  60277 = '60277'
  60278 = '60278'
  60279 = '60279'
  60280 = '60280'
  60281 = '60281'
  60282 = '60282'
  60283 = '60283'
  60284 = '60284'
  60285 = '60285'
  60286 = '60286'
  60287 = '60287'
  60288 = '60288'
  60289 = '60289'
  60290 = '60290'
  60291 = '60291'
  60292 = '60292'
  60293 = '60293'
  60294 = '60294'
  60295 = '60295'
  60296 = '60296'
  60297 = '60297'
  60298 = '60298'
  60299 = '60299'
  60300 = '60300'
  60301 = '60301'
  60302 = '60302'
  60303 = '60303'
  60304 = '60304'
  60305 = '60305'
  60306 = '60306'
  60307 = '60307'
  60308 = '60308'
  60309 = '60309'
  60310 = '60310'
  60311 = '60311'
  60312 = '60312'
  60313 = '60313'
  60314 = '60314'
  60315 = '60315'
  60316 = '60316'
  60317 = '60317'
  60318 = '60318'
  60319 = '60319'
  60320 = '60320'
  60321 = '60321'
  60322 = '60322'
  60323 = '60323'
  60324 = '60324'
  60325 = '60325'
  60326 = '60326'
  60327 = '60327'
  60328 = '60328'
  60329 = '60329'
  60330 = '60330'
  60331 = '60331'
  60332 = '60332'
  60333 = '60333'
  60334 = '60334'
  60335 = '60335'
  60336 = '60336'
  60337 = '60337'
  60338 = '60338'
  60339 = '60339'
  60340 = '60340'
  60341 = '60341'
  60342 = '60342'
  60343 = '60343'
  60344 = '60344'
  60345 = '60345'
  60346 = '60346'
  60347 = '60347'
  60348 = '60348'
  60349 = '60349'
  60350 = '60350'
  60351 = '60351'
  60352 = '60352'
  60353 = '60353'
  60354 = '60354'
  60355 = '60355'
  60356 = '60356'
  60357 = '60357'
  60358 = '60358'
  60359 = '60359'
  60360 = '60360'
  60361 = '60361'
  60362 = '60362'
  60363 = '60363'
  60364 = '60364'
  60365 = '60365'
  60366 = '60366'
  60367 = '60367'
  60368 = '60368'
  60369 = '60369'
  60370 = '60370'
  60371 = '60371'
  60372 = '60372'
  60373 = '60373'
  60374 = '60374'
  60375 = '60375'
  60376 = '60376'
  60377 = '60377'
  60378 = '60378'
  60379 = '60379'
  60380 = '60380'
  60381 = '60381'
  60382 = '60382'
  60383 = '60383'
  60384 = '60384'
  60385 = '60385'
  60386 = '60386'
  60387 = '60387'
  60388 = '60388'
  60389 = '60389'
  60390 = '60390'
  60391 = '60391'
  60392 = '60392'
  60393 = '60393'
  60394 = '60394'
  60395 = '60395'
  60396 = '60396'
  60397 = '60397'
  60398 = '60398'
  60399 = '60399'
  60400 = '60400'
  60401 = '60401'
  60402 = '60402'
  60403 = '60403'
  60404 = '60404'
  60405 = '60405'
  60406 = '60406'
  60407 = '60407'
  60408 = '60408'
  60409 = '60409'
  60410 = '60410'
  60411 = '60411'
  60412 = '60412'
  60413 = '60413'
  60414 = '60414'
  60415 = '60415'
  60416 = '60416'
  60417 = '60417'
  60418 = '60418'
  60419 = '60419'
  60420 = '60420'
  60421 = '60421'
  60422 = '60422'
  60423 = '60423'
  60424 = '60424'
  60425 = '60425'
  60426 = '60426'
  60427 = '60427'
  60428 = '60428'
  60429 = '60429'
  60430 = '60430'
  60431 = '60431'
  60432 = '60432'
  60433 = '60433'
  60434 = '60434'
  60435 = '60435'
  60436 = '60436'
  60437 = '60437'
  60438 = '60438'
  60439 = '60439'
  60440 = '60440'
  60441 = '60441'
  60442 = '60442'
  60443 = '60443'
  60444 = '60444'
  60445 = '60445'
  60446 = '60446'
  60447 = '60447'
  60448 = '60448'
  60449 = '60449'
  60450 = '60450'
  60451 = '60451'
  60452 = '60452'
  60453 = '60453'
  60454 = '60454'
  60455 = '60455'
  60456 = '60456'
  60457 = '60457'
  60458 = '60458'
  60459 = '60459'
  60460 = '60460'
  60461 = '60461'
  60462 = '60462'
  60463 = '60463'
  60464 = '60464'
  60465 = '60465'
  60466 = '60466'
  60467 = '60467'
  60468 = '60468'
  60469 = '60469'
  60470 = '60470'
  60471 = '60471'
  60472 = '60472'
  60473 = '60473'
  60474 = '60474'
  60475 = '60475'
  60476 = '60476'
  60477 = '60477'
  60478 = '60478'
  60479 = '60479'
  60480 = '60480'
  60481 = '60481'
  60482 = '60482'
  60483 = '60483'
  60484 = '60484'
  60485 = '60485'
  60486 = '60486'
  60487 = '60487'
  60488 = '60488'
  60489 = '60489'
  60490 = '60490'
  60491 = '60491'
  60492 = '60492'
  60493 = '60493'
  60494 = '60494'
  60495 = '60495'
  60496 = '60496'
  60497 = '60497'
  60498 = '60498'
  60499 = '60499'
  60500 = '60500'
  60501 = '60501'
  60502 = '60502'
  60503 = '60503'
  60504 = '60504'
  60505 = '60505'
  60506 = '60506'
  60507 = '60507'
  60508 = '60508'
  60509 = '60509'
  60510 = '60510'
  60511 = '60511'
  60512 = '60512'
  60513 = '60513'
  60514 = '60514'
  60515 = '60515'
  60516 = '60516'
  60517 = '60517'
  60518 = '60518'
  60519 = '60519'
  60520 = '60520'
  60521 = '60521'
  60522 = '60522'
  60523 = '60523'
  60524 = '60524'
  60525 = '60525'
  60526 = '60526'
  60527 = '60527'
  60528 = '60528'
  60529 = '60529'
  60530 = '60530'
  60531 = '60531'
  60532 = '60532'
  60533 = '60533'
  60534 = '60534'
  60535 = '60535'
  60536 = '60536'
  60537 = '60537'
  60538 = '60538'
  60539 = '60539'
  60540 = '60540'
  60541 = '60541'
  60542 = '60542'
  60543 = '60543'
  60544 = '60544'
  60545 = '60545'
  60546 = '60546'
  60547 = '60547'
  60548 = '60548'
  60549 = '60549'
  60550 = '60550'
  60551 = '60551'
  60552 = '60552'
  60553 = '60553'
  60554 = '60554'
  60555 = '60555'
  60556 = '60556'
  60557 = '60557'
  60558 = '60558'
  60559 = '60559'
  60560 = '60560'
  60561 = '60561'
  60562 = '60562'
  60563 = '60563'
  60564 = '60564'
  60565 = '60565'
  60566 = '60566'
  60567 = '60567'
  60568 = '60568'
  60569 = '60569'
  60570 = '60570'
  60571 = '60571'
  60572 = '60572'
  60573 = '60573'
  60574 = '60574'
  60575 = '60575'
  60576 = '60576'
  60577 = '60577'
  60578 = '60578'
  60579 = '60579'
  60580 = '60580'
  60581 = '60581'
  60582 = '60582'
  60583 = '60583'
  60584 = '60584'
  60585 = '60585'
  60586 = '60586'
  60587 = '60587'
  60588 = '60588'
  60589 = '60589'
  60590 = '60590'
  60591 = '60591'
  60592 = '60592'
  60593 = '60593'
  60594 = '60594'
  60595 = '60595'
  60596 = '60596'
  60597 = '60597'
  60598 = '60598'
  60599 = '60599'
  60600 = '60600'
  60601 = '60601'
  60602 = '60602'
  60603 = '60603'
  60604 = '60604'
  60605 = '60605'
  60606 = '60606'
  60607 = '60607'
  60608 = '60608'
  60609 = '60609'
  60610 = '60610'
  60611 = '60611'
  60612 = '60612'
  60613 = '60613'
  60614 = '60614'
  60615 = '60615'
  60616 = '60616'
  60617 = '60617'
  60618 = '60618'
  60619 = '60619'
  60620 = '60620'
  60621 = '60621'
  60622 = '60622'
  60623 = '60623'
  60624 = '60624'
  60625 = '60625'
  60626 = '60626'
  60627 = '60627'
  60628 = '60628'
  60629 = '60629'
  60630 = '60630'
  60631 = '60631'
  60632 = '60632'
  60633 = '60633'
  60634 = '60634'
  60635 = '60635'
  60636 = '60636'
  60637 = '60637'
  60638 = '60638'
  60639 = '60639'
  60640 = '60640'
  60641 = '60641'
  60642 = '60642'
  60643 = '60643'
  60644 = '60644'
  60645 = '60645'
  60646 = '60646'
  60647 = '60647'
  60648 = '60648'
  60649 = '60649'
  60650 = '60650'
  60651 = '60651'
  60652 = '60652'
  60653 = '60653'
  60654 = '60654'
  60655 = '60655'
  60656 = '60656'
  60657 = '60657'
  60658 = '60658'
  60659 = '60659'
  60660 = '60660'
  60661 = '60661'
  60662 = '60662'
  60663 = '60663'
  60664 = '60664'
  60665 = '60665'
  60666 = '60666'
  60667 = '60667'
  60668 = '60668'
  60669 = '60669'
  60670 = '60670'
  60671 = '60671'
  60672 = '60672'
  60673 = '60673'
  60674 = '60674'
  60675 = '60675'
  60676 = '60676'
  60677 = '60677'
  60678 = '60678'
  60679 = '60679'
  60680 = '60680'
  60681 = '60681'
  60682 = '60682'
  60683 = '60683'
  60684 = '60684'
  60685 = '60685'
  60686 = '60686'
  60687 = '60687'
  60688 = '60688'
  60689 = '60689'
  60690 = '60690'
  60691 = '60691'
  60692 = '60692'
  60693 = '60693'
  60694 = '60694'
  60695 = '60695'
  60696 = '60696'
  60697 = '60697'
  60698 = '60698'
  60699 = '60699'
  60700 = '60700'
  60701 = '60701'
  60702 = '60702'
  60703 = '60703'
  60704 = '60704'
  60705 = '60705'
  60706 = '60706'
  60707 = '60707'
  60708 = '60708'
  60709 = '60709'
  60710 = '60710'
  60711 = '60711'
  60712 = '60712'
  60713 = '60713'
  60714 = '60714'
  60715 = '60715'
  60716 = '60716'
  60717 = '60717'
  60718 = '60718'
  60719 = '60719'
  60720 = '60720'
  60721 = '60721'
  60722 = '60722'
  60723 = '60723'
  60724 = '60724'
  60725 = '60725'
  60726 = '60726'
  60727 = '60727'
  60728 = '60728'
  60729 = '60729'
  60730 = '60730'
  60731 = '60731'
  60732 = '60732'
  60733 = '60733'
  60734 = '60734'
  60735 = '60735'
  60736 = '60736'
  60737 = '60737'
  60738 = '60738'
  60739 = '60739'
  60740 = '60740'
  60741 = '60741'
  60742 = '60742'
  60743 = '60743'
  60744 = '60744'
  60745 = '60745'
  60746 = '60746'
  60747 = '60747'
  60748 = '60748'
  60749 = '60749'
  60750 = '60750'
  60751 = '60751'
  60752 = '60752'
  60753 = '60753'
  60754 = '60754'
  60755 = '60755'
  60756 = '60756'
  60757 = '60757'
  60758 = '60758'
  60759 = '60759'
  60760 = '60760'
  60761 = '60761'
  60762 = '60762'
  60763 = '60763'
  60764 = '60764'
  60765 = '60765'
  60766 = '60766'
  60767 = '60767'
  60768 = '60768'
  60769 = '60769'
  60770 = '60770'
  60771 = '60771'
  60772 = '60772'
  60773 = '60773'
  60774 = '60774'
  60775 = '60775'
  60776 = '60776'
  60777 = '60777'
  60778 = '60778'
  60779 = '60779'
  60780 = '60780'
  60781 = '60781'
  60782 = '60782'
  60783 = '60783'
  60784 = '60784'
  60785 = '60785'
  60786 = '60786'
  60787 = '60787'
  60788 = '60788'
  60789 = '60789'
  60790 = '60790'
  60791 = '60791'
  60792 = '60792'
  60793 = '60793'
  60794 = '60794'
  60795 = '60795'
  60796 = '60796'
  60797 = '60797'
  60798 = '60798'
  60799 = '60799'
  60800 = '60800'
  60801 = '60801'
  60802 = '60802'
  60803 = '60803'
  60804 = '60804'
  60805 = '60805'
  60806 = '60806'
  60807 = '60807'
  60808 = '60808'
  60809 = '60809'
  60810 = '60810'
  60811 = '60811'
  60812 = '60812'
  60813 = '60813'
  60814 = '60814'
  60815 = '60815'
  60816 = '60816'
  60817 = '60817'
  60818 = '60818'
  60819 = '60819'
  60820 = '60820'
  60821 = '60821'
  60822 = '60822'
  60823 = '60823'
  60824 = '60824'
  60825 = '60825'
  60826 = '60826'
  60827 = '60827'
  60828 = '60828'
  60829 = '60829'
  60830 = '60830'
  60831 = '60831'
  60832 = '60832'
  60833 = '60833'
  60834 = '60834'
  60835 = '60835'
  60836 = '60836'
  60837 = '60837'
  60838 = '60838'
  60839 = '60839'
  60840 = '60840'
  60841 = '60841'
  60842 = '60842'
  60843 = '60843'
  60844 = '60844'
  60845 = '60845'
  60846 = '60846'
  60847 = '60847'
  60848 = '60848'
  60849 = '60849'
  60850 = '60850'
  60851 = '60851'
  60852 = '60852'
  60853 = '60853'
  60854 = '60854'
  60855 = '60855'
  60856 = '60856'
  60857 = '60857'
  60858 = '60858'
  60859 = '60859'
  60860 = '60860'
  60861 = '60861'
  60862 = '60862'
  60863 = '60863'
  60864 = '60864'
  60865 = '60865'
  60866 = '60866'
  60867 = '60867'
  60868 = '60868'
  60869 = '60869'
  60870 = '60870'
  60871 = '60871'
  60872 = '60872'
  60873 = '60873'
  60874 = '60874'
  60875 = '60875'
  60876 = '60876'
  60877 = '60877'
  60878 = '60878'
  60879 = '60879'
  60880 = '60880'
  60881 = '60881'
  60882 = '60882'
  60883 = '60883'
  60884 = '60884'
  60885 = '60885'
  60886 = '60886'
  60887 = '60887'
  60888 = '60888'
  60889 = '60889'
  60890 = '60890'
  60891 = '60891'
  60892 = '60892'
  60893 = '60893'
  60894 = '60894'
  60895 = '60895'
  60896 = '60896'
  60897 = '60897'
  60898 = '60898'
  60899 = '60899'
  60900 = '60900'
  60901 = '60901'
  60902 = '60902'
  60903 = '60903'
  60904 = '60904'
  60905 = '60905'
  60906 = '60906'
  60907 = '60907'
  60908 = '60908'
  60909 = '60909'
  60910 = '60910'
  60911 = '60911'
  60912 = '60912'
  60913 = '60913'
  60914 = '60914'
  60915 = '60915'
  60916 = '60916'
  60917 = '60917'
  60918 = '60918'
  60919 = '60919'
  60920 = '60920'
  60921 = '60921'
  60922 = '60922'
  60923 = '60923'
  60924 = '60924'
  60925 = '60925'
  60926 = '60926'
  60927 = '60927'
  60928 = '60928'
  60929 = '60929'
  60930 = '60930'
  60931 = '60931'
  60932 = '60932'
  60933 = '60933'
  60934 = '60934'
  60935 = '60935'
  60936 = '60936'
  60937 = '60937'
  60938 = '60938'
  60939 = '60939'
  60940 = '60940'
  60941 = '60941'
  60942 = '60942'
  60943 = '60943'
  60944 = '60944'
  60945 = '60945'
  60946 = '60946'
  60947 = '60947'
  60948 = '60948'
  60949 = '60949'
  60950 = '60950'
  60951 = '60951'
  60952 = '60952'
  60953 = '60953'
  60954 = '60954'
  60955 = '60955'
  60956 = '60956'
  60957 = '60957'
  60958 = '60958'
  60959 = '60959'
  60960 = '60960'
  60961 = '60961'
  60962 = '60962'
  60963 = '60963'
  60964 = '60964'
  60965 = '60965'
  60966 = '60966'
  60967 = '60967'
  60968 = '60968'
  60969 = '60969'
  60970 = '60970'
  60971 = '60971'
  60972 = '60972'
  60973 = '60973'
  60974 = '60974'
  60975 = '60975'
  60976 = '60976'
  60977 = '60977'
  60978 = '60978'
  60979 = '60979'
  60980 = '60980'
  60981 = '60981'
  60982 = '60982'
  60983 = '60983'
  60984 = '60984'
  60985 = '60985'
  60986 = '60986'
  60987 = '60987'
  60988 = '60988'
  60989 = '60989'
  60990 = '60990'
  60991 = '60991'
  60992 = '60992'
  60993 = '60993'
  60994 = '60994'
  60995 = '60995'
  60996 = '60996'
  60997 = '60997'
  60998 = '60998'
  60999 = '60999'
  61000 = '61000'
  61001 = '61001'
  61002 = '61002'
  61003 = '61003'
  61004 = '61004'
  61005 = '61005'
  61006 = '61006'
  61007 = '61007'
  61008 = '61008'
  61009 = '61009'
  61010 = '61010'
  61011 = '61011'
  61012 = '61012'
  61013 = '61013'
  61014 = '61014'
  61015 = '61015'
  61016 = '61016'
  61017 = '61017'
  61018 = '61018'
  61019 = '61019'
  61020 = '61020'
  61021 = '61021'
  61022 = '61022'
  61023 = '61023'
  61024 = '61024'
  61025 = '61025'
  61026 = '61026'
  61027 = '61027'
  61028 = '61028'
  61029 = '61029'
  61030 = '61030'
  61031 = '61031'
  61032 = '61032'
  61033 = '61033'
  61034 = '61034'
  61035 = '61035'
  61036 = '61036'
  61037 = '61037'
  61038 = '61038'
  61039 = '61039'
  61040 = '61040'
  61041 = '61041'
  61042 = '61042'
  61043 = '61043'
  61044 = '61044'
  61045 = '61045'
  61046 = '61046'
  61047 = '61047'
  61048 = '61048'
  61049 = '61049'
  61050 = '61050'
  61051 = '61051'
  61052 = '61052'
  61053 = '61053'
  61054 = '61054'
  61055 = '61055'
  61056 = '61056'
  61057 = '61057'
  61058 = '61058'
  61059 = '61059'
  61060 = '61060'
  61061 = '61061'
  61062 = '61062'
  61063 = '61063'
  61064 = '61064'
  61065 = '61065'
  61066 = '61066'
  61067 = '61067'
  61068 = '61068'
  61069 = '61069'
  61070 = '61070'
  61071 = '61071'
  61072 = '61072'
  61073 = '61073'
  61074 = '61074'
  61075 = '61075'
  61076 = '61076'
  61077 = '61077'
  61078 = '61078'
  61079 = '61079'
  61080 = '61080'
  61081 = '61081'
  61082 = '61082'
  61083 = '61083'
  61084 = '61084'
  61085 = '61085'
  61086 = '61086'
  61087 = '61087'
  61088 = '61088'
  61089 = '61089'
  61090 = '61090'
  61091 = '61091'
  61092 = '61092'
  61093 = '61093'
  61094 = '61094'
  61095 = '61095'
  61096 = '61096'
  61097 = '61097'
  61098 = '61098'
  61099 = '61099'
  61100 = '61100'
  61101 = '61101'
  61102 = '61102'
  61103 = '61103'
  61104 = '61104'
  61105 = '61105'
  61106 = '61106'
  61107 = '61107'
  61108 = '61108'
  61109 = '61109'
  61110 = '61110'
  61111 = '61111'
  61112 = '61112'
  61113 = '61113'
  61114 = '61114'
  61115 = '61115'
  61116 = '61116'
  61117 = '61117'
  61118 = '61118'
  61119 = '61119'
  61120 = '61120'
  61121 = '61121'
  61122 = '61122'
  61123 = '61123'
  61124 = '61124'
  61125 = '61125'
  61126 = '61126'
  61127 = '61127'
  61128 = '61128'
  61129 = '61129'
  61130 = '61130'
  61131 = '61131'
  61132 = '61132'
  61133 = '61133'
  61134 = '61134'
  61135 = '61135'
  61136 = '61136'
  61137 = '61137'
  61138 = '61138'
  61139 = '61139'
  61140 = '61140'
  61141 = '61141'
  61142 = '61142'
  61143 = '61143'
  61144 = '61144'
  61145 = '61145'
  61146 = '61146'
  61147 = '61147'
  61148 = '61148'
  61149 = '61149'
  61150 = '61150'
  61151 = '61151'
  61152 = '61152'
  61153 = '61153'
  61154 = '61154'
  61155 = '61155'
  61156 = '61156'
  61157 = '61157'
  61158 = '61158'
  61159 = '61159'
  61160 = '61160'
  61161 = '61161'
  61162 = '61162'
  61163 = '61163'
  61164 = '61164'
  61165 = '61165'
  61166 = '61166'
  61167 = '61167'
  61168 = '61168'
  61169 = '61169'
  61170 = '61170'
  61171 = '61171'
  61172 = '61172'
  61173 = '61173'
  61174 = '61174'
  61175 = '61175'
  61176 = '61176'
  61177 = '61177'
  61178 = '61178'
  61179 = '61179'
  61180 = '61180'
  61181 = '61181'
  61182 = '61182'
  61183 = '61183'
  61184 = '61184'
  61185 = '61185'
  61186 = '61186'
  61187 = '61187'
  61188 = '61188'
  61189 = '61189'
  61190 = '61190'
  61191 = '61191'
  61192 = '61192'
  61193 = '61193'
  61194 = '61194'
  61195 = '61195'
  61196 = '61196'
  61197 = '61197'
  61198 = '61198'
  61199 = '61199'
  61200 = '61200'
  61201 = '61201'
  61202 = '61202'
  61203 = '61203'
  61204 = '61204'
  61205 = '61205'
  61206 = '61206'
  61207 = '61207'
  61208 = '61208'
  61209 = '61209'
  61210 = '61210'
  61211 = '61211'
  61212 = '61212'
  61213 = '61213'
  61214 = '61214'
  61215 = '61215'
  61216 = '61216'
  61217 = '61217'
  61218 = '61218'
  61219 = '61219'
  61220 = '61220'
  61221 = '61221'
  61222 = '61222'
  61223 = '61223'
  61224 = '61224'
  61225 = '61225'
  61226 = '61226'
  61227 = '61227'
  61228 = '61228'
  61229 = '61229'
  61230 = '61230'
  61231 = '61231'
  61232 = '61232'
  61233 = '61233'
  61234 = '61234'
  61235 = '61235'
  61236 = '61236'
  61237 = '61237'
  61238 = '61238'
  61239 = '61239'
  61240 = '61240'
  61241 = '61241'
  61242 = '61242'
  61243 = '61243'
  61244 = '61244'
  61245 = '61245'
  61246 = '61246'
  61247 = '61247'
  61248 = '61248'
  61249 = '61249'
  61250 = '61250'
  61251 = '61251'
  61252 = '61252'
  61253 = '61253'
  61254 = '61254'
  61255 = '61255'
  61256 = '61256'
  61257 = '61257'
  61258 = '61258'
  61259 = '61259'
  61260 = '61260'
  61261 = '61261'
  61262 = '61262'
  61263 = '61263'
  61264 = '61264'
  61265 = '61265'
  61266 = '61266'
  61267 = '61267'
  61268 = '61268'
  61269 = '61269'
  61270 = '61270'
  61271 = '61271'
  61272 = '61272'
  61273 = '61273'
  61274 = '61274'
  61275 = '61275'
  61276 = '61276'
  61277 = '61277'
  61278 = '61278'
  61279 = '61279'
  61280 = '61280'
  61281 = '61281'
  61282 = '61282'
  61283 = '61283'
  61284 = '61284'
  61285 = '61285'
  61286 = '61286'
  61287 = '61287'
  61288 = '61288'
  61289 = '61289'
  61290 = '61290'
  61291 = '61291'
  61292 = '61292'
  61293 = '61293'
  61294 = '61294'
  61295 = '61295'
  61296 = '61296'
  61297 = '61297'
  61298 = '61298'
  61299 = '61299'
  61300 = '61300'
  61301 = '61301'
  61302 = '61302'
  61303 = '61303'
  61304 = '61304'
  61305 = '61305'
  61306 = '61306'
  61307 = '61307'
  61308 = '61308'
  61309 = '61309'
  61310 = '61310'
  61311 = '61311'
  61312 = '61312'
  61313 = '61313'
  61314 = '61314'
  61315 = '61315'
  61316 = '61316'
  61317 = '61317'
  61318 = '61318'
  61319 = '61319'
  61320 = '61320'
  61321 = '61321'
  61322 = '61322'
  61323 = '61323'
  61324 = '61324'
  61325 = '61325'
  61326 = '61326'
  61327 = '61327'
  61328 = '61328'
  61329 = '61329'
  61330 = '61330'
  61331 = '61331'
  61332 = '61332'
  61333 = '61333'
  61334 = '61334'
  61335 = '61335'
  61336 = '61336'
  61337 = '61337'
  61338 = '61338'
  61339 = '61339'
  61340 = '61340'
  61341 = '61341'
  61342 = '61342'
  61343 = '61343'
  61344 = '61344'
  61345 = '61345'
  61346 = '61346'
  61347 = '61347'
  61348 = '61348'
  61349 = '61349'
  61350 = '61350'
  61351 = '61351'
  61352 = '61352'
  61353 = '61353'
  61354 = '61354'
  61355 = '61355'
  61356 = '61356'
  61357 = '61357'
  61358 = '61358'
  61359 = '61359'
  61360 = '61360'
  61361 = '61361'
  61362 = '61362'
  61363 = '61363'
  61364 = '61364'
  61365 = '61365'
  61366 = '61366'
  61367 = '61367'
  61368 = '61368'
  61369 = '61369'
  61370 = '61370'
  61371 = '61371'
  61372 = '61372'
  61373 = '61373'
  61374 = '61374'
  61375 = '61375'
  61376 = '61376'
  61377 = '61377'
  61378 = '61378'
  61379 = '61379'
  61380 = '61380'
  61381 = '61381'
  61382 = '61382'
  61383 = '61383'
  61384 = '61384'
  61385 = '61385'
  61386 = '61386'
  61387 = '61387'
  61388 = '61388'
  61389 = '61389'
  61390 = '61390'
  61391 = '61391'
  61392 = '61392'
  61393 = '61393'
  61394 = '61394'
  61395 = '61395'
  61396 = '61396'
  61397 = '61397'
  61398 = '61398'
  61399 = '61399'
  61400 = '61400'
  61401 = '61401'
  61402 = '61402'
  61403 = '61403'
  61404 = '61404'
  61405 = '61405'
  61406 = '61406'
  61407 = '61407'
  61408 = '61408'
  61409 = '61409'
  61410 = '61410'
  61411 = '61411'
  61412 = '61412'
  61413 = '61413'
  61414 = '61414'
  61415 = '61415'
  61416 = '61416'
  61417 = '61417'
  61418 = '61418'
  61419 = '61419'
  61420 = '61420'
  61421 = '61421'
  61422 = '61422'
  61423 = '61423'
  61424 = '61424'
  61425 = '61425'
  61426 = '61426'
  61427 = '61427'
  61428 = '61428'
  61429 = '61429'
  61430 = '61430'
  61431 = '61431'
  61432 = '61432'
  61433 = '61433'
  61434 = '61434'
  61435 = '61435'
  61436 = '61436'
  61437 = '61437'
  61438 = '61438'
  61439 = '61439'
  61440 = '61440'
  61441 = '61441'
  61442 = '61442'
  61443 = '61443'
  61444 = '61444'
  61445 = '61445'
  61446 = '61446'
  61447 = '61447'
  61448 = '61448'
  61449 = '61449'
  61450 = '61450'
  61451 = '61451'
  61452 = '61452'
  61453 = '61453'
  61454 = '61454'
  61455 = '61455'
  61456 = '61456'
  61457 = '61457'
  61458 = '61458'
  61459 = '61459'
  61460 = '61460'
  61461 = '61461'
  61462 = '61462'
  61463 = '61463'
  61464 = '61464'
  61465 = '61465'
  61466 = '61466'
  61467 = '61467'
  61468 = '61468'
  61469 = '61469'
  61470 = '61470'
  61471 = '61471'
  61472 = '61472'
  61473 = '61473'
  61474 = '61474'
  61475 = '61475'
  61476 = '61476'
  61477 = '61477'
  61478 = '61478'
  61479 = '61479'
  61480 = '61480'
  61481 = '61481'
  61482 = '61482'
  61483 = '61483'
  61484 = '61484'
  61485 = '61485'
  61486 = '61486'
  61487 = '61487'
  61488 = '61488'
  61489 = '61489'
  61490 = '61490'
  61491 = '61491'
  61492 = '61492'
  61493 = '61493'
  61494 = '61494'
  61495 = '61495'
  61496 = '61496'
  61497 = '61497'
  61498 = '61498'
  61499 = '61499'
  61500 = '61500'
  61501 = '61501'
  61502 = '61502'
  61503 = '61503'
  61504 = '61504'
  61505 = '61505'
  61506 = '61506'
  61507 = '61507'
  61508 = '61508'
  61509 = '61509'
  61510 = '61510'
  61511 = '61511'
  61512 = '61512'
  61513 = '61513'
  61514 = '61514'
  61515 = '61515'
  61516 = '61516'
  61517 = '61517'
  61518 = '61518'
  61519 = '61519'
  61520 = '61520'
  61521 = '61521'
  61522 = '61522'
  61523 = '61523'
  61524 = '61524'
  61525 = '61525'
  61526 = '61526'
  61527 = '61527'
  61528 = '61528'
  61529 = '61529'
  61530 = '61530'
  61531 = '61531'
  61532 = '61532'
  61533 = '61533'
  61534 = '61534'
  61535 = '61535'
  61536 = '61536'
  61537 = '61537'
  61538 = '61538'
  61539 = '61539'
  61540 = '61540'
  61541 = '61541'
  61542 = '61542'
  61543 = '61543'
  61544 = '61544'
  61545 = '61545'
  61546 = '61546'
  61547 = '61547'
  61548 = '61548'
  61549 = '61549'
  61550 = '61550'
  61551 = '61551'
  61552 = '61552'
  61553 = '61553'
  61554 = '61554'
  61555 = '61555'
  61556 = '61556'
  61557 = '61557'
  61558 = '61558'
  61559 = '61559'
  61560 = '61560'
  61561 = '61561'
  61562 = '61562'
  61563 = '61563'
  61564 = '61564'
  61565 = '61565'
  61566 = '61566'
  61567 = '61567'
  61568 = '61568'
  61569 = '61569'
  61570 = '61570'
  61571 = '61571'
  61572 = '61572'
  61573 = '61573'
  61574 = '61574'
  61575 = '61575'
  61576 = '61576'
  61577 = '61577'
  61578 = '61578'
  61579 = '61579'
  61580 = '61580'
  61581 = '61581'
  61582 = '61582'
  61583 = '61583'
  61584 = '61584'
  61585 = '61585'
  61586 = '61586'
  61587 = '61587'
  61588 = '61588'
  61589 = '61589'
  61590 = '61590'
  61591 = '61591'
  61592 = '61592'
  61593 = '61593'
  61594 = '61594'
  61595 = '61595'
  61596 = '61596'
  61597 = '61597'
  61598 = '61598'
  61599 = '61599'
  61600 = '61600'
  61601 = '61601'
  61602 = '61602'
  61603 = '61603'
  61604 = '61604'
  61605 = '61605'
  61606 = '61606'
  61607 = '61607'
  61608 = '61608'
  61609 = '61609'
  61610 = '61610'
  61611 = '61611'
  61612 = '61612'
  61613 = '61613'
  61614 = '61614'
  61615 = '61615'
  61616 = '61616'
  61617 = '61617'
  61618 = '61618'
  61619 = '61619'
  61620 = '61620'
  61621 = '61621'
  61622 = '61622'
  61623 = '61623'
  61624 = '61624'
  61625 = '61625'
  61626 = '61626'
  61627 = '61627'
  61628 = '61628'
  61629 = '61629'
  61630 = '61630'
  61631 = '61631'
  61632 = '61632'
  61633 = '61633'
  61634 = '61634'
  61635 = '61635'
  61636 = '61636'
  61637 = '61637'
  61638 = '61638'
  61639 = '61639'
  61640 = '61640'
  61641 = '61641'
  61642 = '61642'
  61643 = '61643'
  61644 = '61644'
  61645 = '61645'
  61646 = '61646'
  61647 = '61647'
  61648 = '61648'
  61649 = '61649'
  61650 = '61650'
  61651 = '61651'
  61652 = '61652'
  61653 = '61653'
  61654 = '61654'
  61655 = '61655'
  61656 = '61656'
  61657 = '61657'
  61658 = '61658'
  61659 = '61659'
  61660 = '61660'
  61661 = '61661'
  61662 = '61662'
  61663 = '61663'
  61664 = '61664'
  61665 = '61665'
  61666 = '61666'
  61667 = '61667'
  61668 = '61668'
  61669 = '61669'
  61670 = '61670'
  61671 = '61671'
  61672 = '61672'
  61673 = '61673'
  61674 = '61674'
  61675 = '61675'
  61676 = '61676'
  61677 = '61677'
  61678 = '61678'
  61679 = '61679'
  61680 = '61680'
  61681 = '61681'
  61682 = '61682'
  61683 = '61683'
  61684 = '61684'
  61685 = '61685'
  61686 = '61686'
  61687 = '61687'
  61688 = '61688'
  61689 = '61689'
  61690 = '61690'
  61691 = '61691'
  61692 = '61692'
  61693 = '61693'
  61694 = '61694'
  61695 = '61695'
  61696 = '61696'
  61697 = '61697'
  61698 = '61698'
  61699 = '61699'
  61700 = '61700'
  61701 = '61701'
  61702 = '61702'
  61703 = '61703'
  61704 = '61704'
  61705 = '61705'
  61706 = '61706'
  61707 = '61707'
  61708 = '61708'
  61709 = '61709'
  61710 = '61710'
  61711 = '61711'
  61712 = '61712'
  61713 = '61713'
  61714 = '61714'
  61715 = '61715'
  61716 = '61716'
  61717 = '61717'
  61718 = '61718'
  61719 = '61719'
  61720 = '61720'
  61721 = '61721'
  61722 = '61722'
  61723 = '61723'
  61724 = '61724'
  61725 = '61725'
  61726 = '61726'
  61727 = '61727'
  61728 = '61728'
  61729 = '61729'
  61730 = '61730'
  61731 = '61731'
  61732 = '61732'
  61733 = '61733'
  61734 = '61734'
  61735 = '61735'
  61736 = '61736'
  61737 = '61737'
  61738 = '61738'
  61739 = '61739'
  61740 = '61740'
  61741 = '61741'
  61742 = '61742'
  61743 = '61743'
  61744 = '61744'
  61745 = '61745'
  61746 = '61746'
  61747 = '61747'
  61748 = '61748'
  61749 = '61749'
  61750 = '61750'
  61751 = '61751'
  61752 = '61752'
  61753 = '61753'
  61754 = '61754'
  61755 = '61755'
  61756 = '61756'
  61757 = '61757'
  61758 = '61758'
  61759 = '61759'
  61760 = '61760'
  61761 = '61761'
  61762 = '61762'
  61763 = '61763'
  61764 = '61764'
  61765 = '61765'
  61766 = '61766'
  61767 = '61767'
  61768 = '61768'
  61769 = '61769'
  61770 = '61770'
  61771 = '61771'
  61772 = '61772'
  61773 = '61773'
  61774 = '61774'
  61775 = '61775'
  61776 = '61776'
  61777 = '61777'
  61778 = '61778'
  61779 = '61779'
  61780 = '61780'
  61781 = '61781'
  61782 = '61782'
  61783 = '61783'
  61784 = '61784'
  61785 = '61785'
  61786 = '61786'
  61787 = '61787'
  61788 = '61788'
  61789 = '61789'
  61790 = '61790'
  61791 = '61791'
  61792 = '61792'
  61793 = '61793'
  61794 = '61794'
  61795 = '61795'
  61796 = '61796'
  61797 = '61797'
  61798 = '61798'
  61799 = '61799'
  61800 = '61800'
  61801 = '61801'
  61802 = '61802'
  61803 = '61803'
  61804 = '61804'
  61805 = '61805'
  61806 = '61806'
  61807 = '61807'
  61808 = '61808'
  61809 = '61809'
  61810 = '61810'
  61811 = '61811'
  61812 = '61812'
  61813 = '61813'
  61814 = '61814'
  61815 = '61815'
  61816 = '61816'
  61817 = '61817'
  61818 = '61818'
  61819 = '61819'
  61820 = '61820'
  61821 = '61821'
  61822 = '61822'
  61823 = '61823'
  61824 = '61824'
  61825 = '61825'
  61826 = '61826'
  61827 = '61827'
  61828 = '61828'
  61829 = '61829'
  61830 = '61830'
  61831 = '61831'
  61832 = '61832'
  61833 = '61833'
  61834 = '61834'
  61835 = '61835'
  61836 = '61836'
  61837 = '61837'
  61838 = '61838'
  61839 = '61839'
  61840 = '61840'
  61841 = '61841'
  61842 = '61842'
  61843 = '61843'
  61844 = '61844'
  61845 = '61845'
  61846 = '61846'
  61847 = '61847'
  61848 = '61848'
  61849 = '61849'
  61850 = '61850'
  61851 = '61851'
  61852 = '61852'
  61853 = '61853'
  61854 = '61854'
  61855 = '61855'
  61856 = '61856'
  61857 = '61857'
  61858 = '61858'
  61859 = '61859'
  61860 = '61860'
  61861 = '61861'
  61862 = '61862'
  61863 = '61863'
  61864 = '61864'
  61865 = '61865'
  61866 = '61866'
  61867 = '61867'
  61868 = '61868'
  61869 = '61869'
  61870 = '61870'
  61871 = '61871'
  61872 = '61872'
  61873 = '61873'
  61874 = '61874'
  61875 = '61875'
  61876 = '61876'
  61877 = '61877'
  61878 = '61878'
  61879 = '61879'
  61880 = '61880'
  61881 = '61881'
  61882 = '61882'
  61883 = '61883'
  61884 = '61884'
  61885 = '61885'
  61886 = '61886'
  61887 = '61887'
  61888 = '61888'
  61889 = '61889'
  61890 = '61890'
  61891 = '61891'
  61892 = '61892'
  61893 = '61893'
  61894 = '61894'
  61895 = '61895'
  61896 = '61896'
  61897 = '61897'
  61898 = '61898'
  61899 = '61899'
  61900 = '61900'
  61901 = '61901'
  61902 = '61902'
  61903 = '61903'
  61904 = '61904'
  61905 = '61905'
  61906 = '61906'
  61907 = '61907'
  61908 = '61908'
  61909 = '61909'
  61910 = '61910'
  61911 = '61911'
  61912 = '61912'
  61913 = '61913'
  61914 = '61914'
  61915 = '61915'
  61916 = '61916'
  61917 = '61917'
  61918 = '61918'
  61919 = '61919'
  61920 = '61920'
  61921 = '61921'
  61922 = '61922'
  61923 = '61923'
  61924 = '61924'
  61925 = '61925'
  61926 = '61926'
  61927 = '61927'
  61928 = '61928'
  61929 = '61929'
  61930 = '61930'
  61931 = '61931'
  61932 = '61932'
  61933 = '61933'
  61934 = '61934'
  61935 = '61935'
  61936 = '61936'
  61937 = '61937'
  61938 = '61938'
  61939 = '61939'
  61940 = '61940'
  61941 = '61941'
  61942 = '61942'
  61943 = '61943'
  61944 = '61944'
  61945 = '61945'
  61946 = '61946'
  61947 = '61947'
  61948 = '61948'
  61949 = '61949'
  61950 = '61950'
  61951 = '61951'
  61952 = '61952'
  61953 = '61953'
  61954 = '61954'
  61955 = '61955'
  61956 = '61956'
  61957 = '61957'
  61958 = '61958'
  61959 = '61959'
  61960 = '61960'
  61961 = '61961'
  61962 = '61962'
  61963 = '61963'
  61964 = '61964'
  61965 = '61965'
  61966 = '61966'
  61967 = '61967'
  61968 = '61968'
  61969 = '61969'
  61970 = '61970'
  61971 = '61971'
  61972 = '61972'
  61973 = '61973'
  61974 = '61974'
  61975 = '61975'
  61976 = '61976'
  61977 = '61977'
  61978 = '61978'
  61979 = '61979'
  61980 = '61980'
  61981 = '61981'
  61982 = '61982'
  61983 = '61983'
  61984 = '61984'
  61985 = '61985'
  61986 = '61986'
  61987 = '61987'
  61988 = '61988'
  61989 = '61989'
  61990 = '61990'
  61991 = '61991'
  61992 = '61992'
  61993 = '61993'
  61994 = '61994'
  61995 = '61995'
  61996 = '61996'
  61997 = '61997'
  61998 = '61998'
  61999 = '61999'
  62000 = '62000'
  62001 = '62001'
  62002 = '62002'
  62003 = '62003'
  62004 = '62004'
  62005 = '62005'
  62006 = '62006'
  62007 = '62007'
  62008 = '62008'
  62009 = '62009'
  62010 = '62010'
  62011 = '62011'
  62012 = '62012'
  62013 = '62013'
  62014 = '62014'
  62015 = '62015'
  62016 = '62016'
  62017 = '62017'
  62018 = '62018'
  62019 = '62019'
  62020 = '62020'
  62021 = '62021'
  62022 = '62022'
  62023 = '62023'
  62024 = '62024'
  62025 = '62025'
  62026 = '62026'
  62027 = '62027'
  62028 = '62028'
  62029 = '62029'
  62030 = '62030'
  62031 = '62031'
  62032 = '62032'
  62033 = '62033'
  62034 = '62034'
  62035 = '62035'
  62036 = '62036'
  62037 = '62037'
  62038 = '62038'
  62039 = '62039'
  62040 = '62040'
  62041 = '62041'
  62042 = '62042'
  62043 = '62043'
  62044 = '62044'
  62045 = '62045'
  62046 = '62046'
  62047 = '62047'
  62048 = '62048'
  62049 = '62049'
  62050 = '62050'
  62051 = '62051'
  62052 = '62052'
  62053 = '62053'
  62054 = '62054'
  62055 = '62055'
  62056 = '62056'
  62057 = '62057'
  62058 = '62058'
  62059 = '62059'
  62060 = '62060'
  62061 = '62061'
  62062 = '62062'
  62063 = '62063'
  62064 = '62064'
  62065 = '62065'
  62066 = '62066'
  62067 = '62067'
  62068 = '62068'
  62069 = '62069'
  62070 = '62070'
  62071 = '62071'
  62072 = '62072'
  62073 = '62073'
  62074 = '62074'
  62075 = '62075'
  62076 = '62076'
  62077 = '62077'
  62078 = '62078'
  62079 = '62079'
  62080 = '62080'
  62081 = '62081'
  62082 = '62082'
  62083 = '62083'
  62084 = '62084'
  62085 = '62085'
  62086 = '62086'
  62087 = '62087'
  62088 = '62088'
  62089 = '62089'
  62090 = '62090'
  62091 = '62091'
  62092 = '62092'
  62093 = '62093'
  62094 = '62094'
  62095 = '62095'
  62096 = '62096'
  62097 = '62097'
  62098 = '62098'
  62099 = '62099'
  62100 = '62100'
  62101 = '62101'
  62102 = '62102'
  62103 = '62103'
  62104 = '62104'
  62105 = '62105'
  62106 = '62106'
  62107 = '62107'
  62108 = '62108'
  62109 = '62109'
  62110 = '62110'
  62111 = '62111'
  62112 = '62112'
  62113 = '62113'
  62114 = '62114'
  62115 = '62115'
  62116 = '62116'
  62117 = '62117'
  62118 = '62118'
  62119 = '62119'
  62120 = '62120'
  62121 = '62121'
  62122 = '62122'
  62123 = '62123'
  62124 = '62124'
  62125 = '62125'
  62126 = '62126'
  62127 = '62127'
  62128 = '62128'
  62129 = '62129'
  62130 = '62130'
  62131 = '62131'
  62132 = '62132'
  62133 = '62133'
  62134 = '62134'
  62135 = '62135'
  62136 = '62136'
  62137 = '62137'
  62138 = '62138'
  62139 = '62139'
  62140 = '62140'
  62141 = '62141'
  62142 = '62142'
  62143 = '62143'
  62144 = '62144'
  62145 = '62145'
  62146 = '62146'
  62147 = '62147'
  62148 = '62148'
  62149 = '62149'
  62150 = '62150'
  62151 = '62151'
  62152 = '62152'
  62153 = '62153'
  62154 = '62154'
  62155 = '62155'
  62156 = '62156'
  62157 = '62157'
  62158 = '62158'
  62159 = '62159'
  62160 = '62160'
  62161 = '62161'
  62162 = '62162'
  62163 = '62163'
  62164 = '62164'
   = ''
END_TEXTLIST

// ---- HMI1/Screens/Dialogs/dialogStation.TcVIS
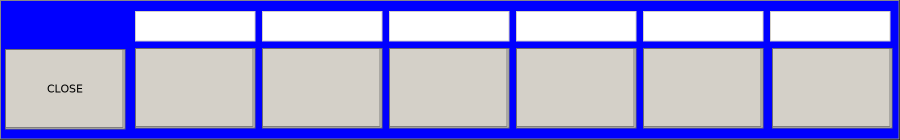
VISUALIZATION dialogStation  // 900x140
    Rectangle (0,0 900x140)
    Group (5,11 887x118)
        Textfield (130,0 120x30), invisible if: NOT gHMIData.gStationEnabled[1], text list: 'ModeStates', text index: S1_Global.station.Data.StationState
        Textfield (257,0 120x30), invisible if: NOT gHMIData.gStationEnabled[2], text list: 'ModeStates', text index: S2_Global.station.Data.StationState
        Textfield (384,0 120x30), invisible if: NOT gHMIData.gStationEnabled[3], text list: 'ModeStates', text index: S3_Global.station.Data.StationState
        Textfield (511,0 120x30), invisible if: NOT gHMIData.gStationEnabled[4], text list: 'ModeStates', text index: S4_Global.station.Data.StationState
        Textfield (638,0 120x30), invisible if: NOT gHMIData.gStationEnabled[5], text list: 'ModeStates', text index: S5_Global.station.Data.StationState
        Textfield (765,0 120x30), invisible if: NOT gHMIData.gStationEnabled[6], text list: 'ModeStates', text index: S6_Global.station.Data.StationState
        Button (130,37 120x80), colour toggle: gHMIData.gStationSelected[1], invisible if: NOT gHMIData.gStationEnabled[1], text list: 'StationNames', text index: 1
            tap gHMIButtons.btnSelectStation1
            OnMouseClick: CloseDialog Dialog=dialogStation, Result=OK, NumpadKeypadSet=True
        Button (257,37 120x80), colour toggle: gHMIData.gStationSelected[2], invisible if: NOT gHMIData.gStationEnabled[2], text list: 'StationNames', text index: 2
            tap gHMIButtons.btnSelectStation2
            OnMouseClick: CloseDialog Dialog=dialogStation, Result=OK, NumpadKeypadSet=True
        Button (384,37 120x80), colour toggle: gHMIData.gStationSelected[3], invisible if: NOT gHMIData.gStationEnabled[3], text list: 'StationNames', text index: 3
            tap gHMIButtons.btnSelectStation3
            OnMouseClick: CloseDialog Dialog=dialogStation, Result=OK, NumpadKeypadSet=True
        Button (511,37 120x80), colour toggle: gHMIData.gStationSelected[4], invisible if: NOT gHMIData.gStationEnabled[4], text list: 'StationNames', text index: 4
            tap gHMIButtons.btnSelectStation4
            OnMouseClick: CloseDialog Dialog=dialogStation, Result=OK, NumpadKeypadSet=True
        Button (638,37 120x80), colour toggle: gHMIData.gStationSelected[5], invisible if: NOT gHMIData.gStationEnabled[5], text list: 'StationNames', text index: 5
            tap gHMIButtons.btnSelectStation5
            OnMouseClick: CloseDialog Dialog=dialogStation, Result=OK, NumpadKeypadSet=True
        Button (767,37 120x80), colour toggle: gHMIData.gStationSelected[6], invisible if: NOT gHMIData.gStationEnabled[6], text list: 'StationNames', text index: 6
            tap gHMIButtons.btnSelectStation6
            OnMouseClick: CloseDialog Dialog=dialogStation, Result=OK, NumpadKeypadSet=True
        Button (0,38 120x80), "CLOSE", colour toggle: gHMIButtons.btnAllStationsSelected, text list: ''
            OnMouseClick: CloseDialog Dialog=dialogStation, Result=None, NumpadKeypadSet=True
END_VISUALIZATION

// ---- HMI1/Templates/MotionRow.TcVIS
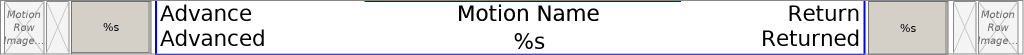
VISUALIZATION MotionRow  // 1024x55
VAR_IN_OUT
	MotionRowInstanceSingle:typeMotionRow; //feedback to motion row to operator
	MotionRowButtonsSingle:typeMotionRowButtons; //button feedback in seperate interface
END_VAR
    Rectangle (155,0 710x55), invisible if: MotionRowInstanceSingle.Returned.bHideCoil AND MotionRowInstanceSingle.bHideName
    Button (868,1 80x55), "%s", text variable: MotionRowInstanceSingle.Returned.NumberOrder, invisible if: MotionRowInstanceSingle.Returned.bHideButton
        tap MotionRowButtonsSingle.btnReturn
        OnMouseDown: execute { gHMIButtons.gAnyButtonPressed := TRUE; }
    Button (71,1 80x53), "%s", text variable: MotionRowInstanceSingle.Advance.NumberOrder, invisible if: MotionRowInstanceSingle.Advance.bHideButton
        tap MotionRowButtonsSingle.btnAdvance
        OnMouseDown: execute { gHMIButtons.gAnyButtonPressed := TRUE; }
    Rectangle (393,25 273x33), "%s", text variable: MotionRowInstanceSingle.strPosn, invisible if: MotionRowInstanceSingle.bHidePosn
        OnMouseClick: OpenDialog Dialog=dialogEnterValue, Parameters={enteredValue: MotionRowButtonsSingle.stnPosnInput}, Selected={1: }, OpenModal=True, OpenCentered=True
    Group (157,1 706x52)
        Rectangle (524,0 182x25), "Return", invisible if: MotionRowInstanceSingle.Returned.bHideCoil or MotionRowInstanceSingle.bIsAbsSymSwitch, text list: 'MotionRowText', text index: MotionRowInstanceSingle.IndexLocation + 3, colour variable: MotionRowInstanceSingle.Returned.CoilColour
        Rectangle (235,0 273x25), "Motion Name", invisible if: MotionRowInstanceSingle.bHideName or MotionRowInstanceSingle.bIsAbsSymSwitch, text list: 'MotionRowText', text index: MotionRowInstanceSingle.IndexLocation + 6
        Rectangle (524,25 182x25), "Returned", invisible if: MotionRowInstanceSingle.Returned.bHideDepth or MotionRowInstanceSingle.bIsAbsSymSwitch, text list: 'MotionRowText', text index: MotionRowInstanceSingle.IndexLocation + 4, colour variable: MotionRowInstanceSingle.Returned.FdbkColour
        Rectangle (0,0 207x25), "Advance", text variable: MotionRowInstanceSingle.Advance.valCoil, invisible if: MotionRowInstanceSingle.Advance.bHideCoil or MotionRowInstanceSingle.bIsAbsSymSwitch, text list: 'MotionRowText', text index: MotionRowInstanceSingle.IndexLocation + 0, colour variable: MotionRowInstanceSingle.Advance.CoilColour
        Rectangle (0,25 207x25), "Advanced", invisible if: MotionRowInstanceSingle.Advance.bHideDepth or MotionRowInstanceSingle.bIsAbsSymSwitch, text list: 'MotionRowText', text index: MotionRowInstanceSingle.IndexLocation + 1, colour variable: MotionRowInstanceSingle.Advance.FdbkColour
    Image (4,1 40x53), invisible if: NOT MotionRowInstanceSingle.Advance.InterlockOK OR MotionRowInstanceSingle.Advance.bHideInterlock, image: MotionRowImages.LeftHighlight
    Image (4,1 40x53), invisible if: MotionRowInstanceSingle.Advance.InterlockOK OR MotionRowInstanceSingle.Advance.bHideInterlock, image: MotionRowImages.LeftNot
    Image (978,1 40x53), invisible if: MotionRowInstanceSingle.Returned.InterlockOK OR MotionRowInstanceSingle.Returned.bHideInterlock, image: MotionRowImages.RightNot
    Image (978,1 40x53), invisible if: NOT MotionRowInstanceSingle.Returned.InterlockOK OR MotionRowInstanceSingle.Returned.bHideInterlock, image: MotionRowImages.RightHighlight
    Image (46,1 23x53), invisible if: MotionRowInstanceSingle.Advance.Prompt OR MotionRowInstanceSingle.Advance.bHidePrompt, image: MotionRowImages.PromptNOK
    Image (953,1 23x53), invisible if: NOT MotionRowInstanceSingle.Returned.Prompt OR MotionRowInstanceSingle.Returned.bHidePrompt, image: MotionRowImages.PromptOK
    Image (953,1 23x53), invisible if: MotionRowInstanceSingle.Returned.Prompt OR MotionRowInstanceSingle.Returned.bHidePrompt, image: MotionRowImages.PromptNOK
    Image (46,1 23x53), invisible if: NOT MotionRowInstanceSingle.Advance.Prompt OR MotionRowInstanceSingle.Advance.bHidePrompt, image: MotionRowImages.PromptOK
    Group (157,1 706x52)
        Rectangle (524,0 182x25), "Return", invisible if: MotionRowInstanceSingle.Returned.bHideCoil or NOT MotionRowInstanceSingle.bIsAbsSymSwitch, text list: 'MotionRowText', text index: MotionRowInstanceSingle.IndexLocation + 3 + 10, colour variable: MotionRowInstanceSingle.Returned.CoilColour
        Rectangle (235,0 273x25), "Motion Name", invisible if: MotionRowInstanceSingle.bHideName or NOT MotionRowInstanceSingle.bIsAbsSymSwitch, text list: 'MotionRowText', text index: MotionRowInstanceSingle.IndexLocation + 6 + 10
        Rectangle (524,25 182x25), "Returned", invisible if: MotionRowInstanceSingle.Returned.bHideDepth or NOT MotionRowInstanceSingle.bIsAbsSymSwitch, text list: 'MotionRowText', text index: MotionRowInstanceSingle.IndexLocation + 4 + 10, colour variable: MotionRowInstanceSingle.Returned.FdbkColour
        Rectangle (0,0 207x25), "Advance", text variable: MotionRowInstanceSingle.Advance.valCoil, invisible if: MotionRowInstanceSingle.Advance.bHideCoil or NOT MotionRowInstanceSingle.bIsAbsSymSwitch, text list: 'MotionRowText', text index: MotionRowInstanceSingle.IndexLocation + 0 + 10, colour variable: MotionRowInstanceSingle.Advance.CoilColour
        Rectangle (0,25 207x25), "Advanced", invisible if: MotionRowInstanceSingle.Advance.bHideDepth or NOT MotionRowInstanceSingle.bIsAbsSymSwitch, text list: 'MotionRowText', text index: MotionRowInstanceSingle.IndexLocation + 1 + 10, colour variable: MotionRowInstanceSingle.Advance.FdbkColour
END_VISUALIZATION

// ---- HMI1/Templates/Tmp_000_Template.TcVIS
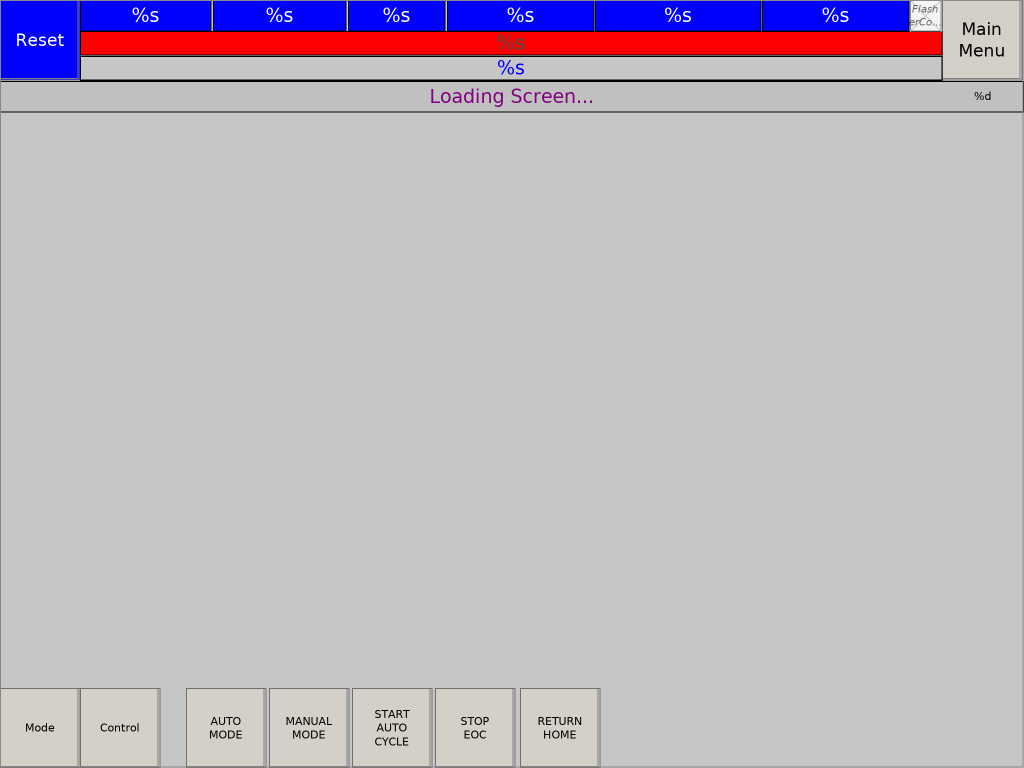
VISUALIZATION Tmp_000_Template  // 1024x768
VAR_IN_OUT
	header:typeHMIheader;
	
END_VAR
    Rectangle (595,0 166x31)
        p2167032090: header.AnyStationWarningColour
    Rectangle (80,57 862x24)
    Group (0,0 1022x80)
        Button (0,0 80x80), "Reset"
            tap gHMIButtons.btnReset
            OnMouseDown: execute { gHMIButtons.gAnyButtonPressed := TRUE; }
        Button (942,0 80x80), "Main Menu"
            OnMouseClick: change screen: Men_030_MenuScreen
            OnMouseDown: execute { gHMIButtons.gAnyButtonPressed := TRUE; }
    Group (80,31 862x24)
        Rectangle (0,0 862x24), "%s", text variable: GlobalMessages.gMsgMc.Warning.topMessage, invisible if: gHMIData.gHideDisplayElementWarningView.McEnabled
        Rectangle (0,0 862x24), "%s", text variable: GlobalMessages.gMsgS1.Warning.topMessage, invisible if: gHMIData.gHideDisplayElementWarningView.S1Enabled
        Rectangle (0,0 862x24), "%s", text variable: GlobalMessages.gMsgS2.Warning.topMessage, invisible if: gHMIData.gHideDisplayElementWarningView.S2Enabled
        Rectangle (0,0 862x24), "%s", text variable: GlobalMessages.gMsgS3.Warning.topMessage, invisible if: gHMIData.gHideDisplayElementWarningView.S3Enabled
        Rectangle (0,0 862x24), "%s", text variable: GlobalMessages.gMsgS4.Warning.topMessage, invisible if: gHMIData.gHideDisplayElementWarningView.S4Enabled
        Rectangle (0,0 862x24), "%s", text variable: GlobalMessages.gMsgS5.Warning.topMessage, invisible if: gHMIData.gHideDisplayElementWarningView.S5Enabled
        Rectangle (0,0 862x24), "%s", text variable: GlobalMessages.gMsgS6.Warning.topMessage, invisible if: gHMIData.gHideDisplayElementWarningView.S6Enabled
    Group (80,31 862x24)
        OnMouseClick: change screen: Msg_020_Alarms
        Rectangle (0,0 862x24), "%s", text variable: GlobalMessages.gMsgMc.Alarm.topMessage, invisible if: gHMIData.gHideDisplayElementAlarmView.McEnabled
        Rectangle (0,0 862x24), "%s", text variable: GlobalMessages.gMsgS1.Alarm.topMessage, invisible if: gHMIData.gHideDisplayElementAlarmView.S1Enabled, text list: ''
        Rectangle (0,0 862x24), "%s", text variable: GlobalMessages.gMsgS2.Alarm.topMessage, invisible if: gHMIData.gHideDisplayElementAlarmView.S2Enabled
        Rectangle (0,0 862x24), "%s", text variable: GlobalMessages.gMsgS3.Alarm.topMessage, invisible if: gHMIData.gHideDisplayElementAlarmView.S3Enabled
        Rectangle (0,0 862x24), "%s", text variable: GlobalMessages.gMsgS4.Alarm.topMessage, invisible if: gHMIData.gHideDisplayElementAlarmView.S4Enabled
        Rectangle (0,0 862x24), "%s", text variable: GlobalMessages.gMsgS5.Alarm.topMessage, invisible if: gHMIData.gHideDisplayElementAlarmView.S5Enabled
        Rectangle (0,0 862x24), "%s", text variable: GlobalMessages.gMsgS6.Alarm.topMessage, invisible if: gHMIData.gHideDisplayElementAlarmView.S6Enabled
    Group (80,56 862x24)
        Rectangle (0,0 862x24), "%s", text variable: GlobalMessages.gMsgS1.Prompts.topMessage, invisible if: gHMIData.gHideDisplayElementPromptView.S1Enabled
        Rectangle (0,0 862x24), "%s", text variable: GlobalMessages.gMsgS2.Prompts.topMessage, invisible if: gHMIData.gHideDisplayElementPromptView.S2Enabled
        Rectangle (0,0 862x24), "%s", text variable: GlobalMessages.gMsgS3.Prompts.topMessage, invisible if: gHMIData.gHideDisplayElementPromptView.S3Enabled
        Rectangle (0,0 862x24), "%s", text variable: GlobalMessages.gMsgS4.Prompts.topMessage, invisible if: gHMIData.gHideDisplayElementPromptView.S4Enabled
        Rectangle (0,0 862x24), "%s", text variable: GlobalMessages.gMsgS5.Prompts.topMessage, invisible if: gHMIData.gHideDisplayElementPromptView.S5Enabled
        Rectangle (0,0 862x24), "%s", text variable: GlobalMessages.gMsgS6.Prompts.topMessage, invisible if: gHMIData.gHideDisplayElementPromptView.S6Enabled
        Rectangle (0,0 862x24), "%s", text variable: GlobalMessages.gMsgMc.Prompts.topMessage, invisible if: gHMIData.gHideDisplayElementPromptView.McEnabled
    Rectangle (0,81 1024x31), "Loading Screen...", text list: 'ScreenNames', text index: gHMIData.gScreenNumber
    Group (0,688 600x80)
        Button (0,0 80x80), "Mode", colour toggle: gHMIButtons.btnFdbk.btnModeFdbk
            OnMouseClick: change screen: Mod_001_ModeScreen
            OnMouseDown: execute { gHMIButtons.gAnyButtonPressed := TRUE; }
        Button (80,0 80x80), "Control", colour toggle: gHMIButtons.btnFdbk.btnControlFdbk
            OnMouseClick: change screen: Previous 
            OnMouseDown: execute { gHMIButtons.gAnyButtonPressed := TRUE; }
        Button (186,0 80x80), "AUTO MODE", colour toggle: gHMIButtons.btnFdbk.btn00Fdbk
            tap gHMIButtons.btnMode.btnFooterAutoMode
            OnMouseDown: execute { gHMIButtons.gAnyButtonPressed := TRUE; }
        Button (269,0 80x80), "MANUAL MODE", colour toggle: gHMIButtons.btnFdbk.btn01Fdbk
            tap gHMIButtons.btnMode.btnFooterManualMode
            OnMouseDown: execute { gHMIButtons.gAnyButtonPressed := TRUE; }
        Button (352,0 80x80), "START AUTO CYCLE", colour toggle: gHMIButtons.btnFdbk.btnAutoCyclingFdbk
            tap gHMIButtons.btnMode.btnFooterAutoCycleStart
            OnMouseDown: execute { gHMIButtons.gAnyButtonPressed := TRUE; }
        Button (435,0 80x80), "STOP EOC", colour toggle: gHMIButtons.btnFdbk.btnIsSEOCFdbk
            tap gHMIButtons.btnMode.btnFooterAutoCycleStopEOC
            OnMouseDown: execute { gHMIButtons.gAnyButtonPressed := TRUE; }
        Button (520,0 80x80), "RETURN HOME", colour toggle: gHMIButtons.btnFdbk.btnIsHomeFdbk
            tap gHMIButtons.btnMode.btnFooterReturnHome
            OnMouseDown: execute { gHMIButtons.gAnyButtonPressed := TRUE; }
    Rectangle (595,0 166x31), "%s", colour toggle: header.AnyStationFaultHeaderActive, invisible if: NOT header.isAnyFaultState, text list: 'AnyStationAlarmList', text index: header.AnyStationFaultHeader
        p2167032090: header.AnyStationFaultColour
    Group (80,0 861x31)
        Rectangle (0,0 131x31), "%s", colour toggle: header.stationstateColour, text list: 'ModeStatesHeader', text index: header.stationstate
        Rectangle (133,0 133x31), "%s", text list: 'CycleType', text index: header.cycleTypeFeedback
        Rectangle (268,0 97x31), "%s", colour toggle: header.isFaultState, text list: 'FaultState', text index: header.FaultStateHeader
        Rectangle (682,0 147x31), "%s", text list: 'StationNames', text index: header.stationNameSelect
            OnMouseClick: OpenDialog Dialog=dialogStation, OpenModal=True, PositionX=100, PositionY=250
        Rectangle (367,0 147x31), "%s", colour toggle: header.homestateColour, text list: 'HomeState', text index: header.homestate
        Image (830,0 31x31), invisible if: header.flasher, image: FlasherCorner.aus
        Image (830,0 31x31), invisible if: NOT header.flasher, image: FlasherCorner.ein
    Rectangle (595,0 166x31), "%s", colour toggle: header.AnyStationWarningHeaderActive, invisible if: NOT header.isAnyWarningState, text list: 'AnyStationWarningList', text index: header.AnyStationWarningHeader
        p2167032090: header.AnyStationWarningColour
    Rectangle (945,81 76x31), "%d", text variable: gHMIData.gScreenNumber
END_VISUALIZATION

// ---- HMI1/Templates/MessageRow.TcVIS
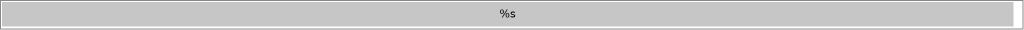
VISUALIZATION MessageRow  // 1024x30
VAR_IN_OUT
	msg:typeMessageRow;
	
	
END_VAR
    Rectangle (2,2 1011x24), "%s", text variable: msg.msgText, colour toggle: msg.isWarning, invisible if: msg.isAlarm, text list: ''
    Rectangle (2,2 1011x24), "%s", text variable: msg.msgText, colour toggle: msg.isAlarm, invisible if: msg.isWarning, text list: ''
END_VISUALIZATION
